// TwinCAT 3 PLC project PLC
// ProgramVersion: 3.1.4024.0
// libraries:
//   Tc2_Standard, * (Beckhoff Automation GmbH)
//   Tc2_System, * (Beckhoff Automation GmbH)
//   Tc3_Module, * (Beckhoff Automation GmbH)
// project tree:
//   / PlcTask.TcTTO
//   POUs/ FB_ConveyorSystem.TcPOU, FB_EmergencyStopState.TcPOU, FB_IdleState.TcPOU, FB_OffState.TcPOU, FB_RunningState.TcPOU, I_State.TcIO, MAIN.TcPOU
// real-time tasks:
//   TASK PlcTask: cycle T#10ms, priority 20, ADS port 350

CONFIGURATION PLC
    RESOURCE PLC ON TwinCAT3
        TASK PlcTask(INTERVAL := T#10ms, PRIORITY := 20);
        PROGRAM MAIN WITH PlcTask : MAIN;
    END_RESOURCE
END_CONFIGURATION

// ---- POUs/I_State.TcIO
INTERFACE I_State

PROPERTY Description : STRING
GET
END_GET
END_PROPERTY

METHOD DetectedPartSensor1 : BOOL
VAR_INPUT
END_VAR
END_METHOD

METHOD DetectedPartSensor2 : BOOL
VAR_INPUT
END_VAR
END_METHOD

METHOD DetectedWeightSensor : BOOL
VAR_INPUT
END_VAR
END_METHOD

METHOD PressEmergencyStop : BOOL
VAR_INPUT
END_VAR
END_METHOD

METHOD PressStart : BOOL
VAR_INPUT
END_VAR
END_METHOD

METHOD PressStop : BOOL
VAR_INPUT
END_VAR
END_METHOD

METHOD ProcessedWeight : BOOL
VAR_INPUT
END_VAR
END_METHOD

END_INTERFACE

// ---- POUs/MAIN.TcPOU
PROGRAM MAIN
VAR
	fbConveyorSystem 		: FB_ConveyorSystem();
	sState 					: STRING;
	nCount 					: INT;
	bPressEmergencyStop 	: BOOL;
	bPressStart 			: BOOL;
	bPressStop 				: BOOL;
	bDetectedPartSensor1 	: BOOL;
	bDetectedWeightSensor 	: BOOL;
	bDetectedPartSensor2 	: BOOL;
END_VAR

fbConveyorSystem(bPressEmergencyStop := bPressEmergencyStop,
				 bPressStart := bPressStart,
				 bPressStop := bPressStop,
				 bDetectedPartSensor1 := bDetectedPartSensor1,
				 bDetectedWeightSensor := bDetectedWeightSensor,
				 bDetectedPartSensor2 := bDetectedPartSensor2);
				 
sState := fbConveyorSystem.ipState.Description;
nCount := fbConveyorSystem.nCount;

bPressEmergencyStop := FALSE;
bPressStart := FALSE;
bPressStop := FALSE;

END_PROGRAM

// ---- POUs/FB_ConveyorSystem.TcPOU
FUNCTION_BLOCK PUBLIC FB_ConveyorSystem
VAR_INPUT
	bPressEmergencyStop : BOOL;
	bPressStart : BOOL;
	bPressStop : BOOL;
	bDetectedPartSensor1: BOOL;
	bDetectedWeightSensor : BOOL;
	bDetectedPartSensor2 : BOOL;
END_VAR
VAR_OUTPUT
	ipState : I_STATE := fbOffState;
	nCount : INT := 0;
	aItemWeights : ARRAY[1..100] OF REAL;
END_VAR
VAR
	fbOffState : FB_OffState(THIS);
	fbIdleState : FB_IdleState(THIS);
	fbRunningState : FB_RunningState(THIS);
	fbEmergencyStopState : FB_EmergencyStopState(THIS);
	
	rtrigPressEmergencyStop : R_TRIG;
	rtrigPressStart : R_TRIG;
	rtrigPressStop : R_TRIG;
	rtrigDetectedPartSensor1 : R_TRIG;
	rtrigDetectedWeightSensor : R_TRIG;
	rtrigProcessedWeight : R_TRIG;
	rtrigDetectedPartSensor2 : R_TRIG;
END_VAR

rtrigPressEmergencyStop(CLK := bPressEmergencyStop);
rtrigPressStart(CLk := bPressStart);
rtrigPressStop(CLK := bPressStop);
rtrigDetectedPartSensor1(CLK := bDetectedPartSensor1);
rtrigDetectedWeightSensor(CLK := bDetectedWeightSensor);
IF (nCount > 0) THEN
	rtrigProcessedWeight(CLK := (aItemWeights[nCount] <> 0));
END_IF
rtrigDetectedPartSensor2(CLK := bDetectedPartSensor2);

IF (rtrigPressEmergencyStop.Q) THEN
	ipState.PressEmergencyStop();
END_IF

IF (rtrigPressStart.Q) THEN
	ipState.PressStart();
END_IF

IF (rtrigPressStop.Q) THEN
	ipState.PressStop();
END_IF

IF (rtrigDetectedPartSensor1.Q) THEN
	ipState.DetectedPartSensor1();
END_IF

IF (rtrigDetectedWeightSensor.Q) THEN
	ipState.DetectedWeightSensor();
END_IF

IF (rtrigProcessedWeight.Q) THEN
	ipState.ProcessedWeight();
END_IF

IF (rtrigDetectedPartSensor2.Q) THEN
	ipState.DetectedPartSensor2();
END_IF

PROPERTY EmergencyStopState : I_STATE
GET
EmergencyStopState := THIS^.fbEmergencyStopState;
END_GET
END_PROPERTY

METHOD FB_init : BOOL
VAR_INPUT
	bInitRetains : BOOL; // if TRUE, the retain variables are initialized (warm start / cold start)
	bInCopyCode : BOOL;  // if TRUE, the instance afterwards gets moved into the copy code (online change
END_VAR
END_METHOD

PROPERTY IdleState : I_STATE
GET
IdleState := THIS^.fbIdleState;
END_GET
END_PROPERTY

PROPERTY OffState : I_STATE
GET
OffState := THIS^.fbOffState;
END_GET
END_PROPERTY

PROPERTY RunningState : I_STATE
GET
RunningState := THIS^.fbRunningState;
END_GET
END_PROPERTY

METHOD SetCount : BOOL
VAR_INPUT
END_VAR
THIS^.nCount := THIS^.nCount + 1;
END_METHOD

METHOD SetState : BOOL
VAR_INPUT
	newState : I_State;
END_VAR
THIS^.ipState := newState;
END_METHOD

METHOD SetWeight : BOOL
VAR_INPUT
	rItemWeight : REAL;
END_VAR
THIS^.aItemWeights[THIS^.nCount] := rItemWeight;
END_METHOD

END_FUNCTION_BLOCK

// ---- POUs/FB_OffState.TcPOU
FUNCTION_BLOCK FB_OffState IMPLEMENTS I_State
VAR_INPUT
END_VAR
VAR_OUTPUT
END_VAR
VAR
	pConveyorSystem : POINTER TO FB_ConveyorSystem;
END_VAR

{warning 'add property implementation'}
PROPERTY Description : STRING
GET
Description := 'Off state';
END_GET
END_PROPERTY

{warning 'add method implementation '}
METHOD DetectedPartSensor1 : BOOL
END_METHOD

{warning 'add method implementation '}
METHOD DetectedPartSensor2 : BOOL
END_METHOD

{warning 'add method implementation '}
METHOD DetectedWeightSensor : BOOL
END_METHOD

METHOD FB_init : BOOL
VAR_INPUT
	bInitRetains : BOOL; // if TRUE, the retain variables are initialized (warm start / cold start)
	bInCopyCode : BOOL;  // if TRUE, the instance afterwards gets moved into the copy code (online change
	pConveyorSystem : POINTER TO FB_ConveyorSystem;
END_VAR
THIS^.pConveyorSystem := pConveyorSystem;
END_METHOD

{warning 'add method implementation '}
METHOD PressEmergencyStop : BOOL
END_METHOD

{warning 'add method implementation '}
METHOD PressStart : BOOL
pConveyorSystem^.SetState(pConveyorSystem^.IdleState);
END_METHOD

{warning 'add method implementation '}
METHOD PressStop : BOOL
END_METHOD

{warning 'add method implementation '}
METHOD ProcessedWeight : BOOL
END_METHOD

END_FUNCTION_BLOCK

// ---- POUs/FB_IdleState.TcPOU
FUNCTION_BLOCK FB_IdleState IMPLEMENTS I_State
VAR_INPUT
END_VAR
VAR_OUTPUT
END_VAR
VAR
	pConveyorSystem : POINTER TO FB_ConveyorSystem;
END_VAR

{warning 'add property implementation'}
PROPERTY Description : STRING
GET
Description := 'Idle state';
END_GET
END_PROPERTY

{warning 'add method implementation '}
METHOD DetectedPartSensor1 : BOOL
THIS^.pConveyorSystem^.SetCount();

IF NOT pConveyorSystem^.bDetectedPartSensor2 THEN
	pConveyorSystem^.SetState(pConveyorSystem^.RunningState);
END_IF
END_METHOD

{warning 'add method implementation '}
METHOD DetectedPartSensor2 : BOOL
END_METHOD

{warning 'add method implementation '}
METHOD DetectedWeightSensor : BOOL
END_METHOD

METHOD FB_init : BOOL
VAR_INPUT
	bInitRetains : BOOL; // if TRUE, the retain variables are initialized (warm start / cold start)
	bInCopyCode : BOOL;  // if TRUE, the instance afterwards gets moved into the copy code (online change)
	pConveyorSystem : POINTER TO FB_ConveyorSystem;
END_VAR
THIS^.pConveyorSystem := pConveyorSystem;
END_METHOD

{warning 'add method implementation '}
METHOD PressEmergencyStop : BOOL
pConveyorSystem^.SetState(pConveyorSystem^.EmergencyStopState);
END_METHOD

{warning 'add method implementation '}
METHOD PressStart : BOOL
END_METHOD

{warning 'add method implementation '}
METHOD PressStop : BOOL
pConveyorSystem^.SetState(pConveyorSystem^.OffState);
END_METHOD

{warning 'add method implementation '}
METHOD ProcessedWeight : BOOL
pConveyorSystem^.SetState(pConveyorSystem^.RunningState);
END_METHOD

END_FUNCTION_BLOCK

// ---- POUs/FB_RunningState.TcPOU
FUNCTION_BLOCK FB_RunningState IMPLEMENTS I_State
VAR_INPUT
END_VAR
VAR_OUTPUT
END_VAR
VAR
	pConveyorSystem : POINTER TO FB_ConveyorSystem;
END_VAR

{warning 'add property implementation'}
PROPERTY Description : STRING
GET
Description := 'Running state';
END_GET
END_PROPERTY

{warning 'add method implementation '}
METHOD DetectedPartSensor1 : BOOL
END_METHOD

{warning 'add method implementation '}
METHOD DetectedPartSensor2 : BOOL
pConveyorSystem^.SetState(pConveyorSystem^.IdleState);
END_METHOD

{warning 'add method implementation '}
METHOD DetectedWeightSensor : BOOL
VAR
	fWeight : REAL;
	fbRandomNumber : DRAND;
END_VAR
IF pConveyorSystem^.aItemWeights[pConveyorSystem^.nCount] = 0 THEN
	pConveyorSystem^.SetState(pConveyorSystem^.IdleState);
	fbRandomNumber(SEED := 1, Num => fWeight);
	fWeight := fWeight * 1000 + 5.0;
	pConveyorSystem^.SetWeight(fWeight);
END_IF
END_METHOD

METHOD FB_init : BOOL
VAR_INPUT
	bInitRetains : BOOL; // if TRUE, the retain variables are initialized (warm start / cold start)
	bInCopyCode : BOOL;  // if TRUE, the instance afterwards gets moved into the copy code (online change)
	pConveyorSystem : POINTER TO FB_ConveyorSystem;
END_VAR
THIS^.pConveyorSystem := pConveyorSystem;
END_METHOD

{warning 'add method implementation '}
METHOD PressEmergencyStop : BOOL
pConveyorSystem^.SetState(pConveyorSystem^.EmergencyStopState);
END_METHOD

{warning 'add method implementation '}
METHOD PressStart : BOOL
END_METHOD

{warning 'add method implementation '}
METHOD PressStop : BOOL
END_METHOD

{warning 'add method implementation '}
METHOD ProcessedWeight : BOOL
END_METHOD

END_FUNCTION_BLOCK

// ---- POUs/FB_EmergencyStopState.TcPOU
FUNCTION_BLOCK FB_EmergencyStopState IMPLEMENTS I_State
VAR_INPUT
END_VAR
VAR_OUTPUT
END_VAR
VAR
	pConveyorSystem : POINTER TO FB_ConveyorSystem;
END_VAR

{warning 'add property implementation'}
PROPERTY Description : STRING
GET
END_GET
END_PROPERTY

{warning 'add method implementation '}
METHOD DetectedPartSensor1 : BOOL
END_METHOD

{warning 'add method implementation '}
METHOD DetectedPartSensor2 : BOOL
END_METHOD

{warning 'add method implementation '}
METHOD DetectedWeightSensor : BOOL
END_METHOD

METHOD FB_init : BOOL
VAR_INPUT
	bInitRetains : BOOL; // if TRUE, the retain variables are initialized (warm start / cold start)
	bInCopyCode : BOOL;  // if TRUE, the instance afterwards gets moved into the copy code (online change)
	pConveyorSystem : POINTER TO FB_ConveyorSystem;
END_VAR
THIS^.pConveyorSystem := pConveyorSystem;
END_METHOD

{warning 'add method implementation '}
METHOD PressEmergencyStop : BOOL
END_METHOD

{warning 'add method implementation '}
METHOD PressStart : BOOL
END_METHOD

{warning 'add method implementation '}
METHOD PressStop : BOOL
END_METHOD

{warning 'add method implementation '}
METHOD ProcessedWeight : BOOL
END_METHOD

END_FUNCTION_BLOCK
